(* IEC 61131-3 sources: programs/VI-54/VI-54_20171205/VI-54_20171205/Stations/PLC_VI54/VI-54_171014/Class/FcTeach, 1 file *)

(* ---- FcTeach.st ---- *)
(*!
<Class
	Name               = "FcTeach"
	Revision           = "0.0"
	RealtimeTask       = "false"
	CyclicTask         = "true"
	DefCyclictime      = "cCT"
	BackgroundTask     = "false"
	Sigmatek           = "false"
	OSInterface        = "false"
	HighPriority       = "false"
	Automatic          = "false"
	UpdateMode         = "Prescan"
	SharedCommandTable = "true"
	Objectsize         = "(570,240)">
	<Channels>
		<Server Name="Comm" Visualized="true" Initialize="false" WriteProtected="false" Retentive="false"/>
		<Server Name="FcState" Visualized="true" Initialize="false" WriteProtected="true" Retentive="false"/>
		<Server Name="TeachState" Visualized="true" Initialize="false" WriteProtected="true" Retentive="false"/>
		<Client Name="iState" Required="true" Internal="false"/>
		<Client Name="oTeach" Required="true" Internal="false"/>
	</Channels>
</Class>
*)
FcTeach : CLASS
  //Servers:
	Comm 	: SvrChCmd_DINT;
	FcState 	: SvrCh_DINT;
	TeachState 	: SvrCh_TeachEnum;
  //Clients:
	iState 	: CltCh_DINT;
	oTeach 	: CltCh_DINT;
  //Variables:
		TmrTeach 	: UDINT;
  //Functions:

	FUNCTION VIRTUAL GLOBAL CyWork
		VAR_INPUT
			EAX 	: UDINT;
		END_VAR
		VAR_OUTPUT
			state (EAX) 	: UDINT;
		END_VAR;
  //Tables:
	FUNCTION @STD
		VAR_OUTPUT
			ret_code	: CONFSTATES;
		END_VAR;
	FUNCTION GLOBAL TAB @CT_;
END_CLASS;

FUNCTION VIRTUAL GLOBAL FcTeach::CyWork
	VAR_INPUT
		EAX 	: UDINT;
	END_VAR
	VAR_OUTPUT
		state (EAX) 	: UDINT;
	END_VAR

  iState := iState.Read();
  FcState := iState;

  case TeachState of
  TeachIdel:
    oTeach := 0;
    if Comm = 1 then
      TmrTeach := ops.tAbsolute;
      TeachState := Teaching;
    elsif Comm = 2 then
      TmrTeach := ops.tAbsolute;
      TeachState := TeachMode;
    end_if;

  Teaching:
    oTeach := 1;
    if ops.tAbsolute - TmrTeach >= 1500 then  // switching to teach mode
      TmrTeach := ops.tAbsolute;
      TeachState := TeachingReady;
    end_if;

  TeachMode:
    oTeach := 1;
    if ops.tAbsolute - TmrTeach >= 11000 then // switching teaching mode
      TmrTeach := ops.tAbsolute;
      TeachState := TeachingReady;
    end_if;

  TeachingReady:
    oTeach := 0;
    if ops.tAbsolute - TmrTeach >= 1000 then
      TmrTeach := ops.tAbsolute;
      Comm := 0;
      TeachState := TeachIdel;
    end_if;

  end_case;

  oTeach.Write (oTeach);

	state := READY;

END_FUNCTION
